PROGRAM prgEM
VAR
	FB_Phoenix:FB_PhoenixContact_EM_EEM_EM375;
	
	lrPower_Grid_TotalkW			: LREAL;			//{#lynus.ag#()}
	lrPower_Grid_L1				: LREAL;			//{#lynus.ag#()}
	lrPower_Grid_L2				: LREAL;			//{#lynus.ag#()}
	lrPower_Grid_L3				: LREAL;			//{#lynus.ag#()}
	lrCurrent_Grid_L1			: LREAL;			//{#lynus.ag#()}
	lrCurrent_Grid_L2			: LREAL;			//{#lynus.ag#()}
	lrCurrent_Grid_L3			: LREAL;			//{#lynus.ag#()}
	lrVoltage_Grid_L1N			: LREAL;			//{#lynus.ag#()}
	lrVoltage_Grid_L2N			: LREAL;			//{#lynus.ag#()}
	lrVoltage_Grid_L3N			: LREAL;			//{#lynus.ag#()}
	

	flEMPowerTotal		: LREAL;
	bPullSuccessfull 	: BOOL;
	udintErrorID		: UDINT;


	uint_State								AT%I* 	: uint;
	lrPower_House_kW			: LREAL;			//{#lynus.ag#()}
		
END_VAR

VAR PERSISTENT
	bEnableEM			: 	BOOL;
END_VAR


// lrPower_House_kW := LIMIT(0,lrPower_Grid_TotalkW - prgCS1.lrPower_Alfen_1_S1 + prgPV.lrPower_PV_kW,100);


FB_Phoenix(
	bEnable:= TRUE, 
	byUnitID:= 255, 
	sIPAdress:= '192.168.1.11', 
	stDataEMPower=> , 
	stDataEMCounter=> , 
	stDataEMPowerRealTime=> , 
	stDataEMCounterRealTime=> , 
	diNrOfEM_OUT=> );

lrPower_Grid_TotalkW 	:= 	FB_Phoenix.stDataEMPower.lrPowerTotal;
lrPower_Grid_L1		 	:= 	FB_Phoenix.stDataEMPower.lrPowerL1;
lrPower_Grid_L2		 	:= 	FB_Phoenix.stDataEMPower.lrPowerL2;
lrPower_Grid_L3		 	:= 	FB_Phoenix.stDataEMPower.lrPowerL3;
lrCurrent_Grid_L1 		:= 	FB_Phoenix.stDataEMPower.lrCurrentL1;
lrCurrent_Grid_L2 		:= 	FB_Phoenix.stDataEMPower.lrCurrentL2;
lrCurrent_Grid_L3 		:= 	FB_Phoenix.stDataEMPower.lrCurrentL3;
lrVoltage_Grid_L1N		:= 	FB_Phoenix.stDataEMPower.lrVoltageL1N;
lrVoltage_Grid_L2N		:= 	FB_Phoenix.stDataEMPower.lrVoltageL2N;
lrVoltage_Grid_L3N		:= 	FB_Phoenix.stDataEMPower.lrVoltageL3N;

END_PROGRAM

(* stored: Version 1.1.0.1, ProductVersion 3.1.4024.12
   POU prgEM: Id {2e582916-7d77-4864-9d3b-f8d4d01a814d}, SpecialFunc None *)
